TYPE ST_Motion :
STRUCT
	fbFirstMotor			:FB_Motor;
END_STRUCT
END_TYPE

(* stored: Version 1.1.0.1, ProductVersion 3.1.4024.12
   DUT ST_Motion: Id {95a81582-6ab9-43f6-952b-e0e898d718e8} *)
